(* Logix 5000 project; controller RG_Chopper vendor 1 type 14 code 235 rev 32.12; software revision 32.04; part 4 of 6 *)
(* tags used below, declared in another part *)
   L2_FAIL_TMR : TIMER;   // LSSL2 Fail Always Open Detect
   LSSL2_FAIL : BOOL;   // Lower Safety Limit Switch LSS-L2 Fail
   LSSL2_FAIL2 : BOOL;   // Lower Safety Limit Switch LSS-L2 Mode 2
   LSSU2_FAIL : BOOL;   // Upper Safety Limit Switch LSS-U2 Fail
   LSSU2_FAIL2 : BOOL;   // Upper Safety Limit Switch USS-L2 Mode 2
   U2_FAIL_TMR : TIMER;   // LSSU2 Fail Always Open Detect
   _DBL101_TANK_LEVEL : BOOL;   // Conentrate Chopper Level Switch Local:1:I.Data.9
   ALARM_FATAL : BOOL;   // Fatal Alarm Stops All Operation
   ALARM_GATE_OPEN : BOOL;   // Gate Open
   AUTO_ALL : BOOL;   // All Devices to AUTO
   CB104_DUMPER_AUX : BOOL;   // CB104 Dumper Aux From Dumper Control
   CIP_CMPLT : BOOL;   // CIP Complete Indicator
   CYC_CIP : BOOL;   // CIP Cycle Running
   CYC_RUN : BOOL;   // Production Cycle Running
   DBT101 : TD_TA_TP_8PORT_IOL;   // DTT101 Hot Water Temperature IO-Link RAW
   DBT102 : TD_TA_TP_8PORT_IOL;   // DBT102 Product Temperature IO-Link RAW
   DBX101_AM : PUSH_PUSH_PB;   // DBX-101 Push-Push Button Control
   DBX101_AUX : BOOL;   // DBX-101 Agitator Motor Aux
   DBX101_CTL : HOA_CTRL_v2;   // DBX-101 Agitator Motor Control Block
   DBX101_FAULT : BOOL;
   DBX101_MAN : PUSH_PUSH_PB;   // DBX-101 Manual Run Push-Push
   DBX101_OL : BOOL;   // DBX-101 Motor OverLoad Status
   DBX101_START : BOOL;   // DBX-101 Agitator Start Safety Mapped DBX101_S_START
   DBX102_AM : PUSH_PUSH_PB;   // DBX-102 Push-Push Button Control
   DBX102_AUX : ALIAS FOR SIGNAL_IN_RG_CHOPPER.0;   // DBX-102 VFD Active AUX
   DBX102_CTL : HOA_CTRL_v2;   // DBX102 Product Discharge Pump Control Block
   DBX102_FAULT : BOOL;   // DBX-102 Discharge Pump Drive Fault
   DBX102_M_FAULT : BOOL;   // DBX-102 Discharge Pump Drive or Motor Fault
   DBX102_MAN : PUSH_PUSH_PB;   // DBX-102 Manual Control Push-Push
   DBX102_START : BOOL;   // DBX-102 Product Pump VFD START
   DBX103_AM : PUSH_PUSH_PB;   // DBX-103 Push-Push Button Control
   DBX103_AUX : BOOL;   // DBX-103 Water Pump Aux
   DBX103_CTL : HOA_CTRL_v2;   // DBX-103 Hot Water Pump Control Block
   DBX103_FAULT : BOOL;   // DBX-103 Hot Water Pump Fault
   DBX103_MAN : PUSH_PUSH_PB;   // DBX-103 Manual Run Push-Push
   DBX103_OL : BOOL;   // DBX-103 Motor OverLoad Status
   DBX103_START : BOOL;   // DBX-103 Water Pump Start Safety Mapped DBX103_S_START
   DBX104_AM : PUSH_PUSH_PB;   // DBX-104 Push-Push Button Control
   DBX104_AUX : BOOL;   // DBX-104 VFD Active AUX
   DBX104_CTL : HOA_CTRL_v2;   // DBX-104 Reversing Motor Starter Control
   DBX104_DD : PUSH_PUSH_PB;   // DBX104 VFD Direction DOWN Control
   DBX104_DU : PUSH_PUSH_PB;   // DBX104 VFD Direction UP Control
   DBX104_DWN : BOOL;   // DBX-104 Drum Dumper VFD Direction DOWN
   DBX104_FAULT : BOOL;   // DBX-104 Dumper Elevator Drive Fault
   DBX104_M_FAULT : BOOL;   // DBX-104 Dumper Elevator Drive or Motor Fault
   DBX104_MAN : PUSH_PUSH_PB;   // DBX-104 Manual Control Push-Push
   DBX104_START : BOOL;   // DBX-104 Drum Dumper VFD START
   DBX104_UP : BOOL;   // DBX-104 Drum Dumper VFD Direction UP
   DLT101 : PN_PI_PP_8PORT_IOL;   // DLT101 Tank Level IO-Link RAW
   DLT101_LVL_SCL : REAL;   // Tank Level Scaled (0.0 - 100.0%)
   DLT101_SCL : ANLG_SCALE;   // Tank Level Scaling Block
   DLT101_Tk : TK_CTRL;   // Tank Level Control
   DTT101 : REAL;   // DTT-101 Hot Water Temperature Analong In
   DTT102 : REAL;   // Discharge Product Temperature
   DWN_MKBK : BOOL;   // Elevator Down Make / Break LS_L1 Detection
   DWN_MKBK1 : BOOL;   // Elevator Down Make / Break Memory 1
   DWN_STP : BOOL;   // Elevator Down STOP
   Fault_ACK : BOOL;   // Fault Acknowledge
   FAULT_ACK_PB : BOOL;   // Fault ACK Push Button
   Gate_SW1 : DCI_MONITOR;   // Safety Switch Gate_SW1 SW105 A/B
   Gate_SW2 : DCI_MONITOR;   // Safety Switch Gate_SW2 SW108 A/B
   LEVEL_TIMER : TIMER;   // Juice Tank At High Level
   LOT1_TMR : TIMER;   // Lower Over Travel Switch Disable Timer
   LS_L1 : BOOL;   // New Dumper LOWER Limit Switch #1
   LS_LID_OPN : BOOL;   // Lid Open Switch IO-Link Master Mapped X04
   LS_M1 : BOOL;   // New Dumper MIDDLE Limit Switch #1
   LS_U1 : BOOL;   // New Dumper UPPER Limit Switch #1
   LSS_L2 : BOOL;   // New Dumper LOWER Safety Limit Switch #2
   LSS_LOT1 : BOOL;   // New Dumper LOWER OVER TRAVEL Limit Switch
   LSS_U2 : BOOL;   // New Dumper UPPER Safety Limit Switch #2
   ONESHOT : DINT;   // One-shot Word
   PB101 : BOOL;   // Drum Dumper Elevator UP Push Button
   PB102 : BOOL;   // Drum Dumper Elevator DOWN Push Button
   PB103 : BOOL;   // Drum Dumper Elevator STOP Push Button
   PROC_TMR : TIMER[16];   // Process Timers
   S_ESTOP : BOOL;   // Safety ESTOP
   S_Fault_Res : BOOL;   // Safety Circuit Fault Reset
   S_SW_IN : DINT;   // Safety Switch Input Array
   SCR1291 : BOOL;   // Dumper Estop Permissive Lost SCR-1291
   SHTDWN_ACTV : BOOL;   // System Shutdown is In Progress
   SHTDWN_CMPLT : BOOL;   // System Shutdown Complete
   SHUTDOWN : DINT;   // System Shutdown Control Bits
   SIGNAL_OUT_RG_CHOPPER : DINT;
   SPARE_IN : DINT;   // Spare Input
   STARTUP : DINT;   // System Startup Control Bits
   STOP_ALL : BOOL;   // Stop All
   SW101_START_PB : BOOL;   // Start PB HMI
   SW102_STOP_PB : BOOL;   // Stop PB HMI
   SW103_CIP_PB : BOOL;   // CIP PB HMI
   SW104_ESTOP : BOOL;   // Safety E-Stop SW-104
   SW105_DEBOUNCE : TIMER;   // SW-105 Gate Switch Debounce Timer
   SW105_GATE_SWITCH : BOOL;   // Safety Switch Gate SW #1 SW105 A/B
   SW106_LC : LIGHT_CURTAIN;   // Safety SW106 Light Curain
   SW106_LIGHT_CUR : BOOL;   // Safety Light Curtain SW-106
   SW107_TANK_LID : BOOL;   // Tank Lid Safety Switch Active
   SW108_DEBOUNCE : TIMER;   // SW-108 Gate Switch Debounce Timer
   SW108_GATE_SWITCH : BOOL;   // Safety Switch Gate SW #2 SW108 A/B
   SW109 : BOOL;   // Drum Dumper Upper Limit Switch
   SW110 : BOOL;   // Drum Dumper Lower Limit Switch
   Tank_Lid1 : EMERGENCY_STOP;   // Safety Switch Tank Lid Status SW105 A/B
   TP3232_TMP_1_Scaled : REAL;   // Hot Water Temperature Scaled
   TP3232_TMP_2_Scaled : REAL;   // Product Temperature Scaled
   UP_MKBK : BOOL;   // Elevator Down Make / Break LS_U1 Detection
   UP_MKBK1 : BOOL;   // Elevator Up Make / Break Memory 1
   UP_STP : BOOL;   // Elevator Up STOP
(* MainProgram, continued *)

ROUTINE InLink   (* ladder *)
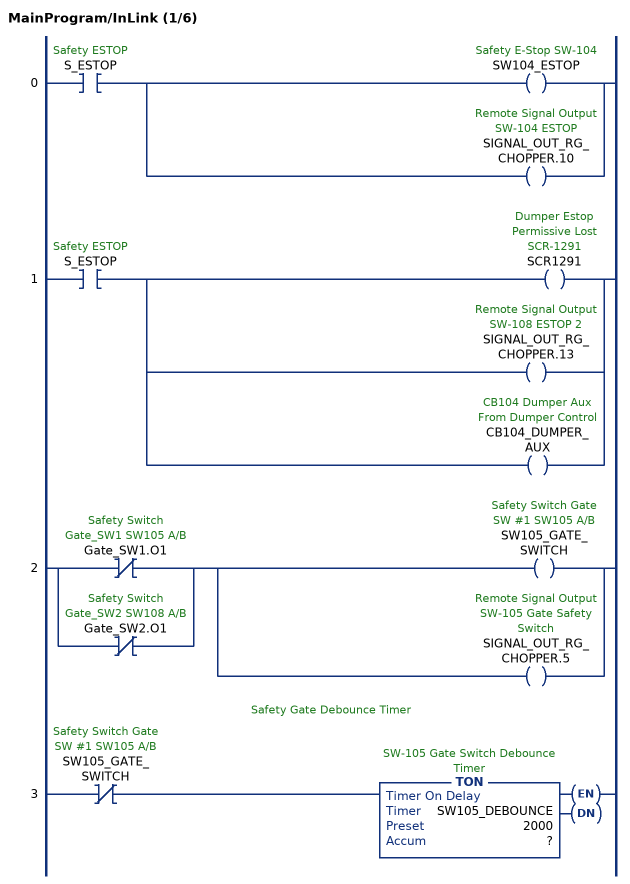
   0: XIC(S_ESTOP)[OTE(SW104_ESTOP) ,OTE(SIGNAL_OUT_RG_CHOPPER.10) ];
   1: XIC(S_ESTOP)[OTE(SCR1291) ,OTE(SIGNAL_OUT_RG_CHOPPER.13) ,OTE(CB104_DUMPER_AUX) ];
   2: [XIO(Gate_SW1.O1) ,XIO(Gate_SW2.O1) ][OTE(SW105_GATE_SWITCH) ,OTE(SIGNAL_OUT_RG_CHOPPER.5) ];
   // Safety Gate Debounce Timer
   3: XIO(SW105_GATE_SWITCH)TON(SW105_DEBOUNCE,?,?);
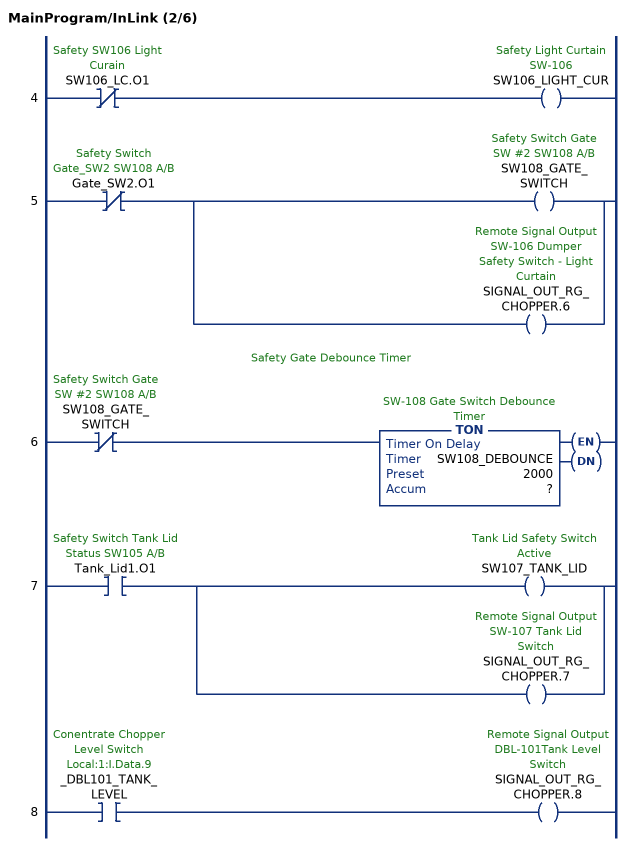
   4: XIO(SW106_LC.O1)OTE(SW106_LIGHT_CUR);
   5: XIO(Gate_SW2.O1)[OTE(SW108_GATE_SWITCH) ,OTE(SIGNAL_OUT_RG_CHOPPER.6) ];
   // Safety Gate Debounce Timer
   6: XIO(SW108_GATE_SWITCH)TON(SW108_DEBOUNCE,?,?);
   7: XIC(Tank_Lid1.O1)[OTE(SW107_TANK_LID) ,OTE(SIGNAL_OUT_RG_CHOPPER.7) ];
   8: XIC(_DBL101_TANK_LEVEL)OTE(SIGNAL_OUT_RG_CHOPPER.8);
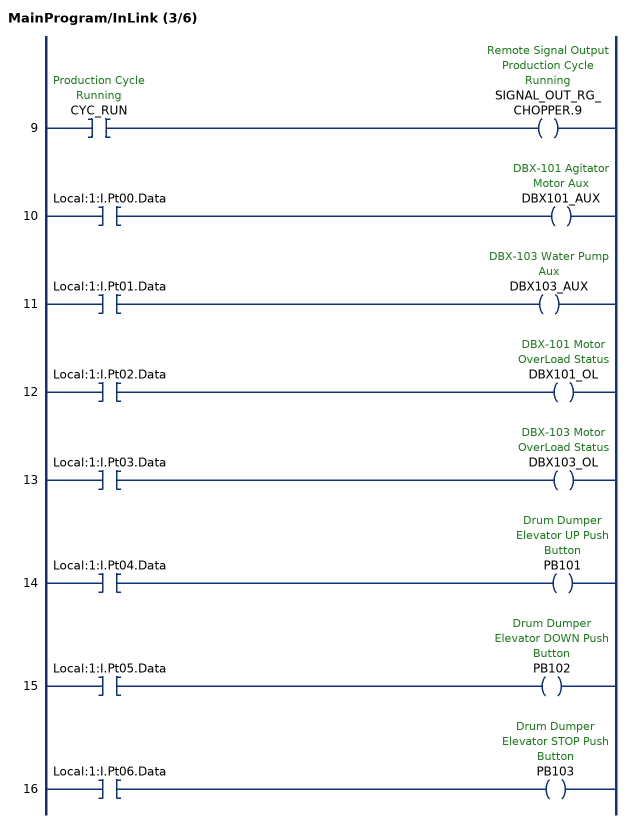
   9: XIC(CYC_RUN)OTE(SIGNAL_OUT_RG_CHOPPER.9);
   10: XIC(Local:1:I.Pt00.Data)OTE(DBX101_AUX);
   11: XIC(Local:1:I.Pt01.Data)OTE(DBX103_AUX);
   12: XIC(Local:1:I.Pt02.Data)OTE(DBX101_OL);
   13: XIC(Local:1:I.Pt03.Data)OTE(DBX103_OL);
   14: XIC(Local:1:I.Pt04.Data)OTE(PB101);
   15: XIC(Local:1:I.Pt05.Data)OTE(PB102);
   16: XIC(Local:1:I.Pt06.Data)OTE(PB103);
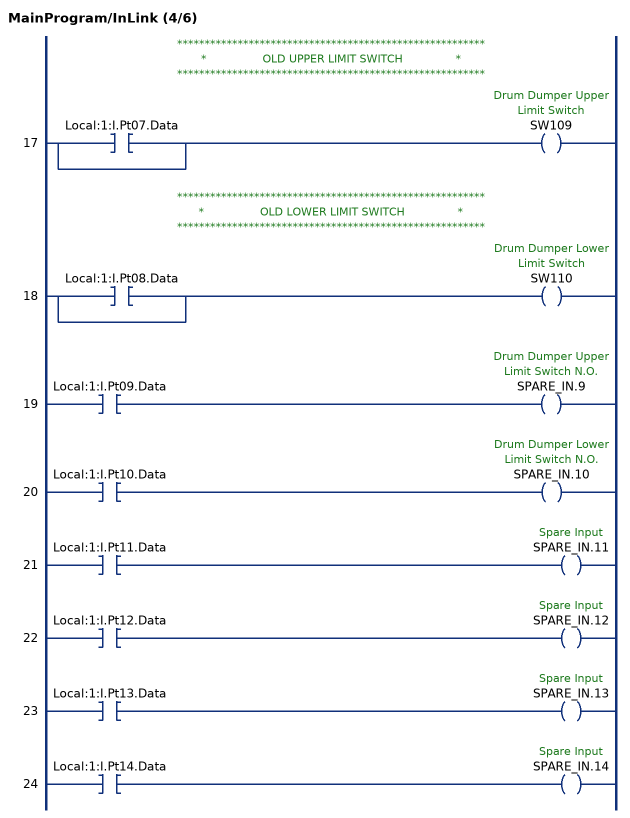
   // ********************************************************
   // *                OLD UPPER LIMIT SWITCH               *
   // ********************************************************
   17: [XIC(Local:1:I.Pt07.Data) ,]OTE(SW109);
   // ********************************************************
   // *                OLD LOWER LIMIT SWITCH               *
   // ********************************************************
   18: [XIC(Local:1:I.Pt08.Data) ,]OTE(SW110);
   19: XIC(Local:1:I.Pt09.Data)OTE(SPARE_IN.9);
   20: XIC(Local:1:I.Pt10.Data)OTE(SPARE_IN.10);
   21: XIC(Local:1:I.Pt11.Data)OTE(SPARE_IN.11);
   22: XIC(Local:1:I.Pt12.Data)OTE(SPARE_IN.12);
   23: XIC(Local:1:I.Pt13.Data)OTE(SPARE_IN.13);
   24: XIC(Local:1:I.Pt14.Data)OTE(SPARE_IN.14);
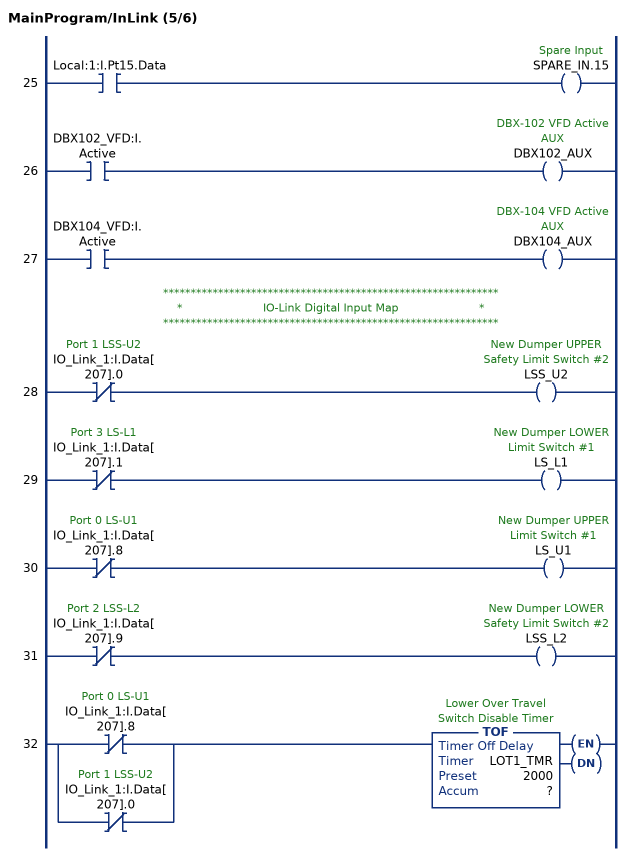
   25: XIC(Local:1:I.Pt15.Data)OTE(SPARE_IN.15);
   26: XIC(DBX102_VFD:I.Active)OTE(DBX102_AUX);
   27: XIC(DBX104_VFD:I.Active)OTE(DBX104_AUX);
   // *************************************************************
   // *                       IO-Link Digital Input Map                       *
   // *************************************************************
   28: XIO(IO_Link_1:I.Data[207].0)OTE(LSS_U2);
   29: XIO(IO_Link_1:I.Data[207].1)OTE(LS_L1);
   30: XIO(IO_Link_1:I.Data[207].8)OTE(LS_U1);
   31: XIO(IO_Link_1:I.Data[207].9)OTE(LSS_L2);
   32: [XIO(IO_Link_1:I.Data[207].8) ,XIO(IO_Link_1:I.Data[207].0) ]TOF(LOT1_TMR,?,?);
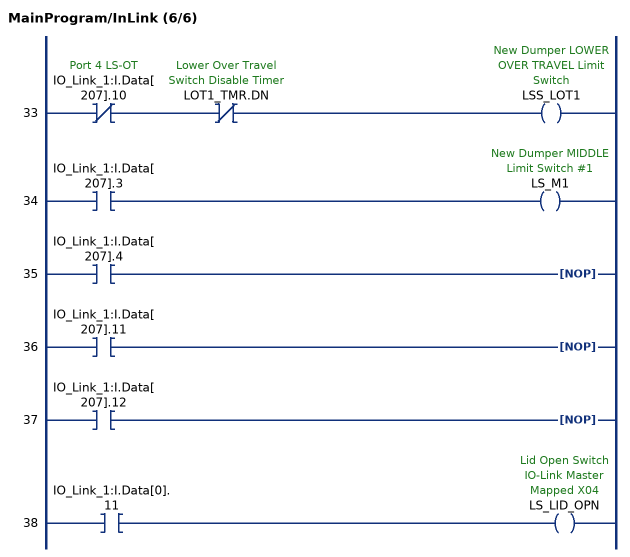
   33: XIO(IO_Link_1:I.Data[207].10)XIO(LOT1_TMR.DN)OTE(LSS_LOT1);
   34: XIC(IO_Link_1:I.Data[207].3)OTE(LS_M1);
   35: XIC(IO_Link_1:I.Data[207].4)NOP();
   36: XIC(IO_Link_1:I.Data[207].11)NOP();
   37: XIC(IO_Link_1:I.Data[207].12)NOP();
   38: XIC(IO_Link_1:I.Data[0].11)OTE(LS_LID_OPN);
END_ROUTINE

ROUTINE IO_Link   (* ladder *)
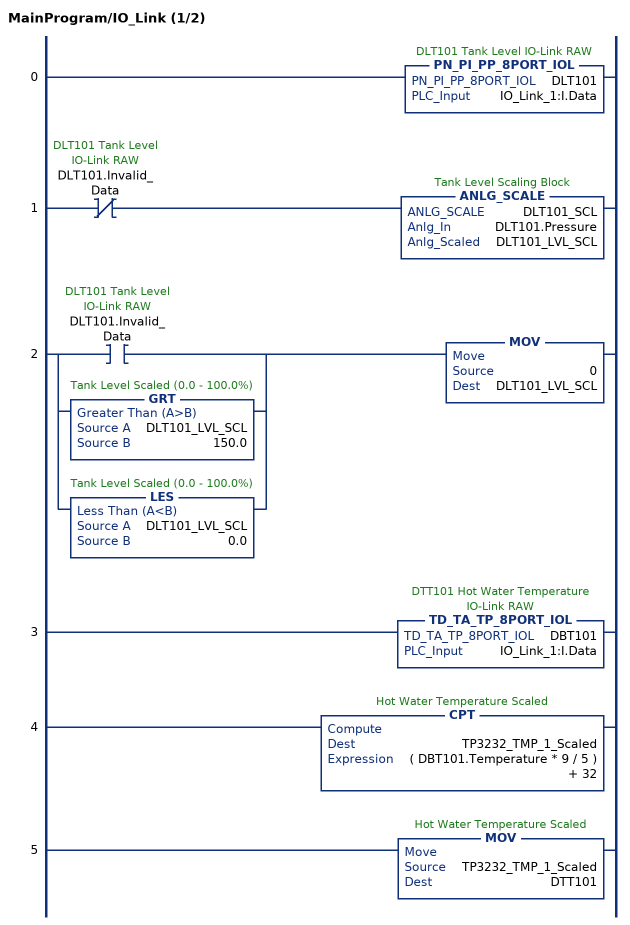
   0: PN_PI_PP_8PORT_IOL(DLT101,IO_Link_1:I.Data);
   1: XIO(DLT101.Invalid_Data)ANLG_SCALE(DLT101_SCL,DLT101.Pressure,DLT101_LVL_SCL);
   2: [XIC(DLT101.Invalid_Data) ,GRT(DLT101_LVL_SCL,150.0) ,LES(DLT101_LVL_SCL,0.0) ]MOV(0,DLT101_LVL_SCL);
   3: TD_TA_TP_8PORT_IOL(DBT101,IO_Link_1:I.Data);
   4: CPT(TP3232_TMP_1_Scaled,( DBT101.Temperature * 9 / 5 ) + 32);
   5: MOV(TP3232_TMP_1_Scaled,DTT101);
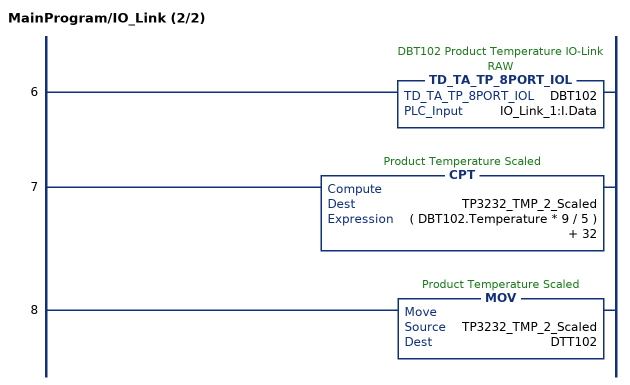
   6: TD_TA_TP_8PORT_IOL(DBT102,IO_Link_1:I.Data);
   7: CPT(TP3232_TMP_2_Scaled,( DBT102.Temperature * 9 / 5 ) + 32);
   8: MOV(TP3232_TMP_2_Scaled,DTT102);
END_ROUTINE

ROUTINE LOGIC   (* ladder *)
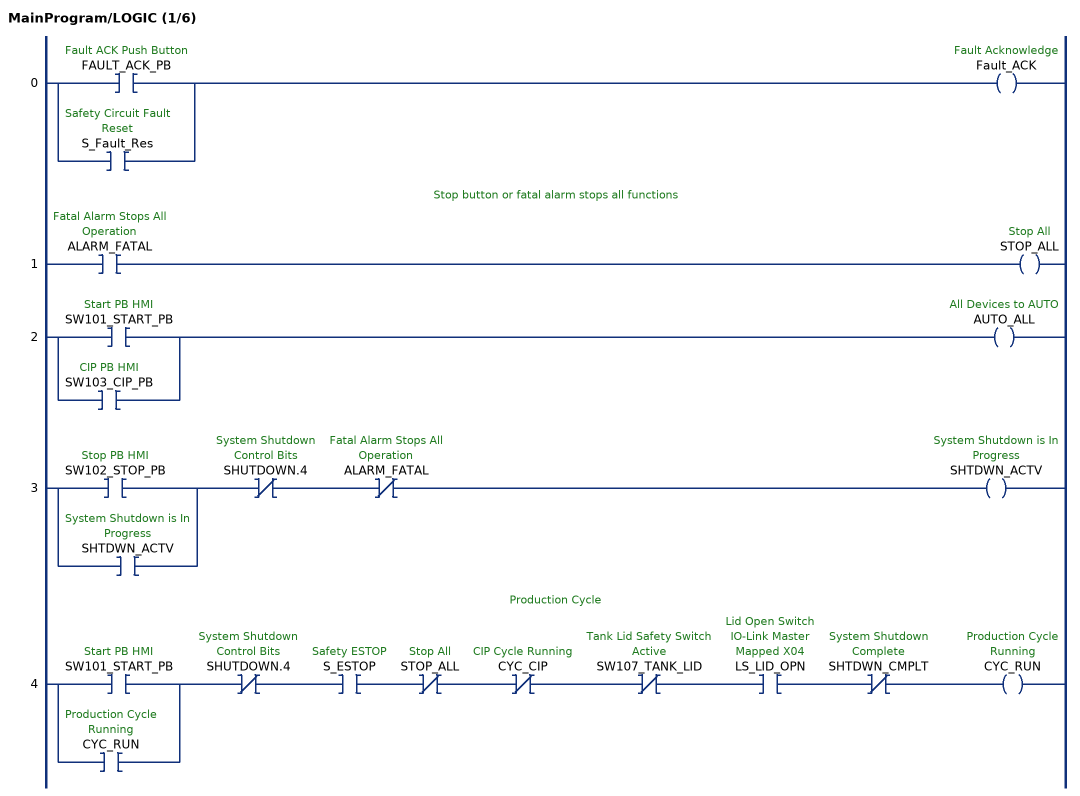
   0: [XIC(FAULT_ACK_PB) ,XIC(S_Fault_Res) ]OTE(Fault_ACK);
   // Stop button or fatal alarm stops all functions
   1: XIC(ALARM_FATAL)OTE(STOP_ALL);
   2: [XIC(SW101_START_PB) ,XIC(SW103_CIP_PB) ]OTE(AUTO_ALL);
   3: [XIC(SW102_STOP_PB) ,XIC(SHTDWN_ACTV) ]XIO(SHUTDOWN.4)XIO(ALARM_FATAL)OTE(SHTDWN_ACTV);
   // Production Cycle
   4: [XIC(SW101_START_PB) ,XIC(CYC_RUN) ]XIO(SHUTDOWN.4)XIC(S_ESTOP)XIO(STOP_ALL)XIO(CYC_CIP)XIO(SW107_TANK_LID)XIC(LS_LID_OPN)XIO(SHTDWN_CMPLT)OTE(CYC_RUN);
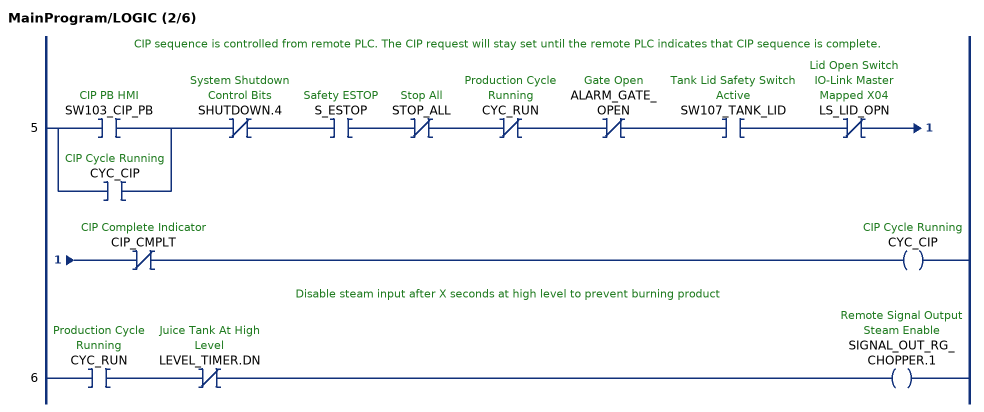
   // CIP sequence is controlled from remote PLC. The CIP request will stay set until the remote PLC indicates that CIP sequence is complete.
   5: [XIC(SW103_CIP_PB) ,XIC(CYC_CIP) ]XIO(SHUTDOWN.4)XIC(S_ESTOP)XIO(STOP_ALL)XIO(CYC_RUN)XIO(ALARM_GATE_OPEN)XIC(SW107_TANK_LID)XIO(LS_LID_OPN)XIO(CIP_CMPLT)OTE(CYC_CIP);
   // Disable steam input after X seconds at high level to prevent burning product
   6: XIC(CYC_RUN)XIO(LEVEL_TIMER.DN)OTE(SIGNAL_OUT_RG_CHOPPER.1);
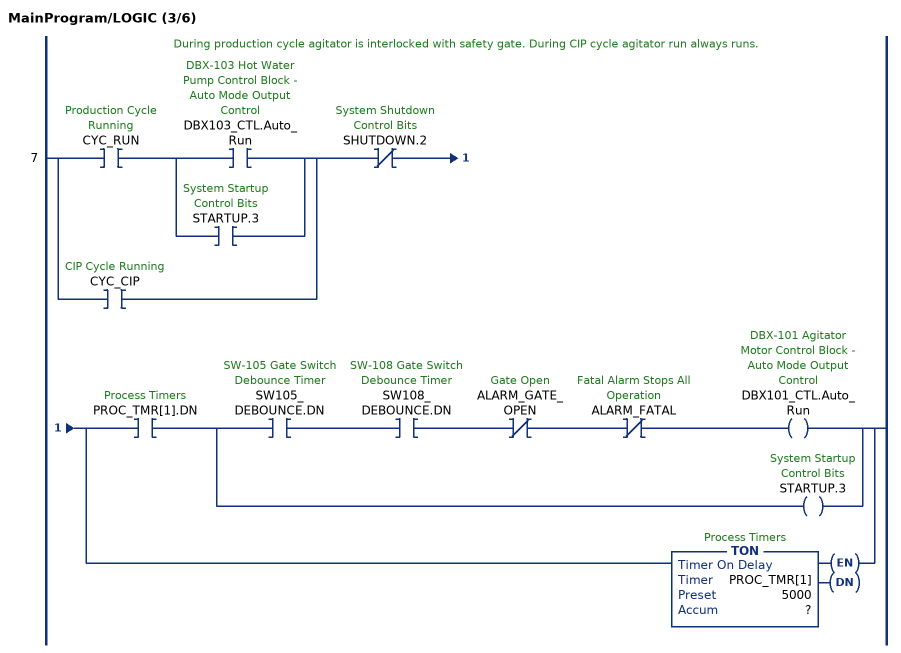
   // During production cycle agitator is interlocked with safety gate. During CIP cycle agitator run always runs.
   7: [XIC(CYC_RUN) [XIC(DBX103_CTL.Auto_Run) ,XIC(STARTUP.3) ] ,XIC(CYC_CIP) ]XIO(SHUTDOWN.2)[XIC(PROC_TMR[1].DN) [XIC(SW105_DEBOUNCE.DN) XIC(SW108_DEBOUNCE.DN) XIO(ALARM_GATE_OPEN) XIO(ALARM_FATAL) OTE(DBX101_CTL.Auto_Run) ,OTE(STARTUP.3) ] ,TON(PROC_TMR[1],?,?) ];
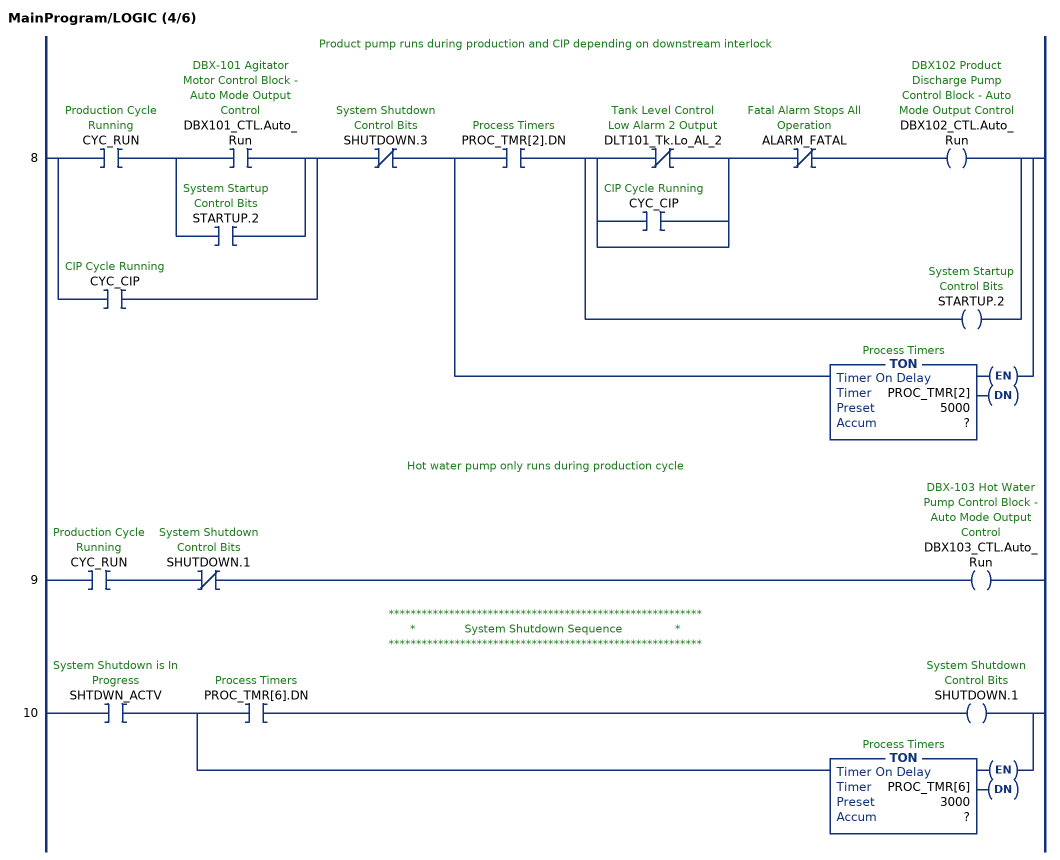
   // Product pump runs during production and CIP depending on downstream interlock
   8: [XIC(CYC_RUN) [XIC(DBX101_CTL.Auto_Run) ,XIC(STARTUP.2) ] ,XIC(CYC_CIP) ]XIO(SHUTDOWN.3)[XIC(PROC_TMR[2].DN) [[XIO(DLT101_Tk.Lo_AL_2) ,XIC(CYC_CIP) ,] XIO(ALARM_FATAL) OTE(DBX102_CTL.Auto_Run) ,OTE(STARTUP.2) ] ,TON(PROC_TMR[2],?,?) ];
   // Hot water pump only runs during production cycle
   9: XIC(CYC_RUN)XIO(SHUTDOWN.1)OTE(DBX103_CTL.Auto_Run);
   // *********************************************************
   // *              System Shutdown Sequence               *
   // *********************************************************
   10: XIC(SHTDWN_ACTV)[XIC(PROC_TMR[6].DN) OTE(SHUTDOWN.1) ,TON(PROC_TMR[6],?,?) ];
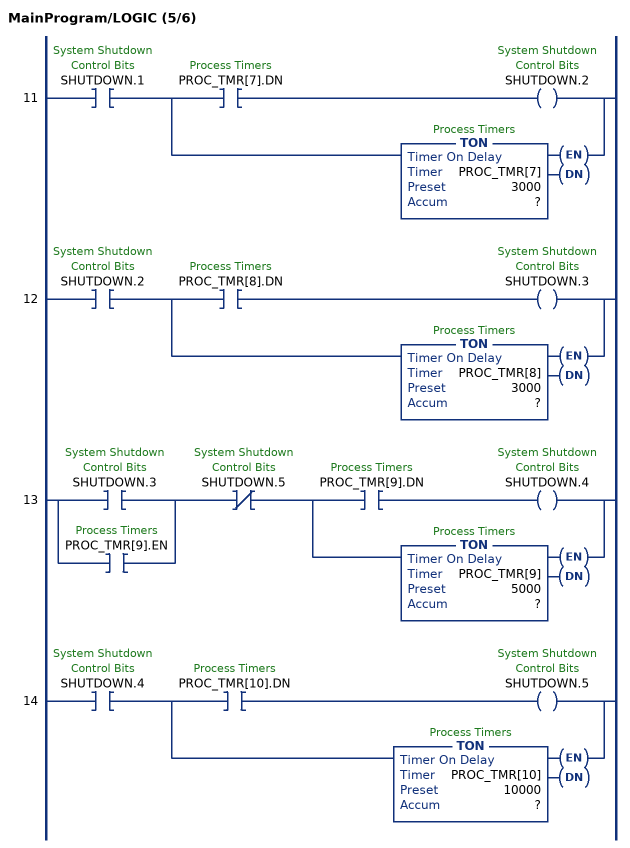
   11: XIC(SHUTDOWN.1)[XIC(PROC_TMR[7].DN) OTE(SHUTDOWN.2) ,TON(PROC_TMR[7],?,?) ];
   12: XIC(SHUTDOWN.2)[XIC(PROC_TMR[8].DN) OTE(SHUTDOWN.3) ,TON(PROC_TMR[8],?,?) ];
   13: [XIC(SHUTDOWN.3) ,XIC(PROC_TMR[9].EN) ]XIO(SHUTDOWN.5)[XIC(PROC_TMR[9].DN) OTE(SHUTDOWN.4) ,TON(PROC_TMR[9],?,?) ];
   14: XIC(SHUTDOWN.4)[XIC(PROC_TMR[10].DN) OTE(SHUTDOWN.5) ,TON(PROC_TMR[10],?,?) ];
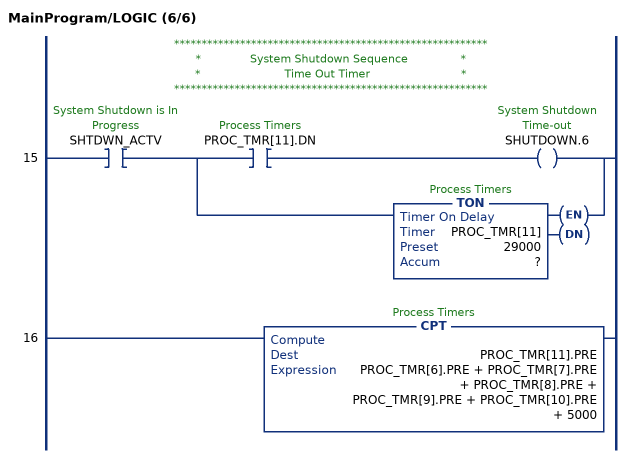
   // *********************************************************
   // *              System Shutdown Sequence               *
   // *                        Time Out Timer                          *
   // *********************************************************
   15: XIC(SHTDWN_ACTV)[XIC(PROC_TMR[11].DN) OTE(SHUTDOWN.6) ,TON(PROC_TMR[11],?,?) ];
   16: CPT(PROC_TMR[11].PRE,PROC_TMR[6].PRE + PROC_TMR[7].PRE + PROC_TMR[8].PRE + PROC_TMR[9].PRE + PROC_TMR[10].PRE + 5000);
END_ROUTINE

ROUTINE MainRoutine   (* ladder *)
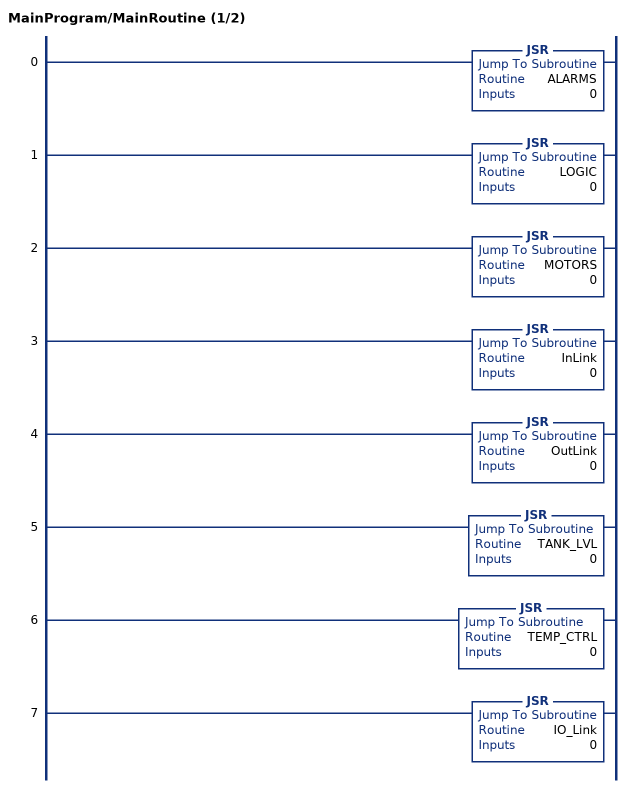
   0: JSR(ALARMS,0);
   1: JSR(LOGIC,0);
   2: JSR(MOTORS,0);
   3: JSR(InLink,0);
   4: JSR(OutLink,0);
   5: JSR(TANK_LVL,0);
   6: JSR(TEMP_CTRL,0);
   7: JSR(IO_Link,0);
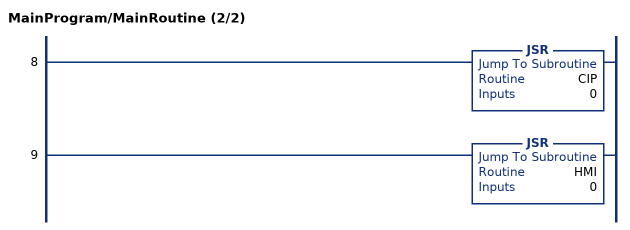
   8: JSR(CIP,0);
   9: JSR(HMI,0);
END_ROUTINE

ROUTINE MOTORS   (* ladder *)
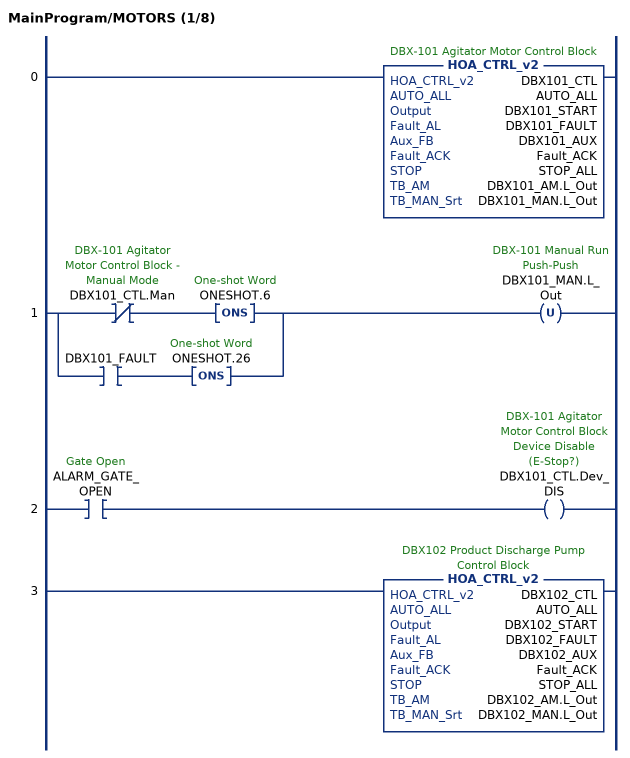
   0: HOA_CTRL_v2(DBX101_CTL,AUTO_ALL,DBX101_START,DBX101_FAULT,DBX101_AUX,Fault_ACK,STOP_ALL,DBX101_AM.L_Out,DBX101_MAN.L_Out);
   1: [XIO(DBX101_CTL.Man) ONS(ONESHOT.6) ,XIC(DBX101_FAULT) ONS(ONESHOT.26) ]OTU(DBX101_MAN.L_Out);
   2: XIC(ALARM_GATE_OPEN)OTE(DBX101_CTL.Dev_DIS);
   3: HOA_CTRL_v2(DBX102_CTL,AUTO_ALL,DBX102_START,DBX102_FAULT,DBX102_AUX,Fault_ACK,STOP_ALL,DBX102_AM.L_Out,DBX102_MAN.L_Out);
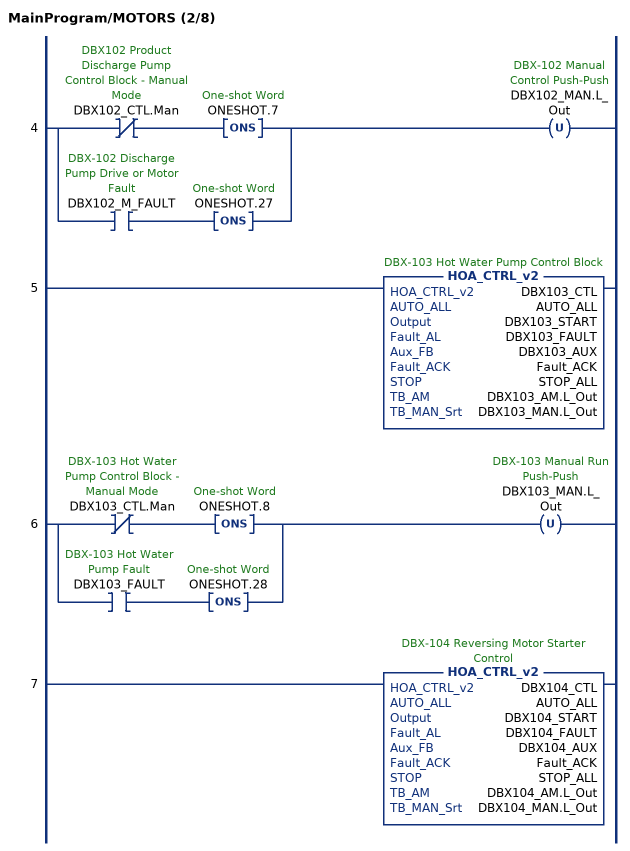
   4: [XIO(DBX102_CTL.Man) ONS(ONESHOT.7) ,XIC(DBX102_M_FAULT) ONS(ONESHOT.27) ]OTU(DBX102_MAN.L_Out);
   5: HOA_CTRL_v2(DBX103_CTL,AUTO_ALL,DBX103_START,DBX103_FAULT,DBX103_AUX,Fault_ACK,STOP_ALL,DBX103_AM.L_Out,DBX103_MAN.L_Out);
   6: [XIO(DBX103_CTL.Man) ONS(ONESHOT.8) ,XIC(DBX103_FAULT) ONS(ONESHOT.28) ]OTU(DBX103_MAN.L_Out);
   7: HOA_CTRL_v2(DBX104_CTL,AUTO_ALL,DBX104_START,DBX104_FAULT,DBX104_AUX,Fault_ACK,STOP_ALL,DBX104_AM.L_Out,DBX104_MAN.L_Out);
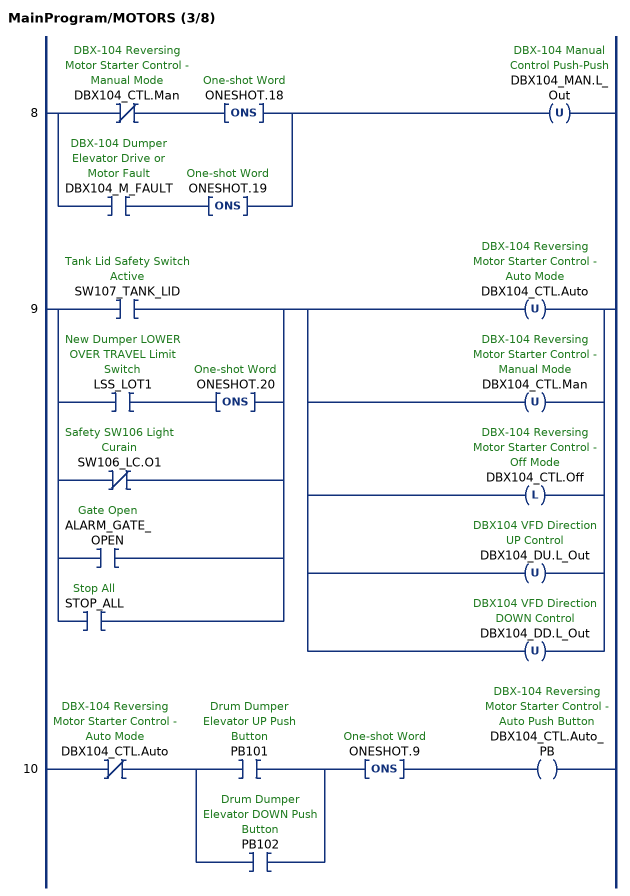
   8: [XIO(DBX104_CTL.Man) ONS(ONESHOT.18) ,XIC(DBX104_M_FAULT) ONS(ONESHOT.19) ]OTU(DBX104_MAN.L_Out);
   9: [XIC(SW107_TANK_LID) ,XIC(LSS_LOT1) ONS(ONESHOT.20) ,XIO(SW106_LC.O1) ,XIC(ALARM_GATE_OPEN) ,XIC(STOP_ALL) ][OTU(DBX104_CTL.Auto) ,OTU(DBX104_CTL.Man) ,OTL(DBX104_CTL.Off) ,OTU(DBX104_DU.L_Out) ,OTU(DBX104_DD.L_Out) ];
   10: XIO(DBX104_CTL.Auto)[XIC(PB101) ,XIC(PB102) ]ONS(ONESHOT.9)OTE(DBX104_CTL.Auto_PB);
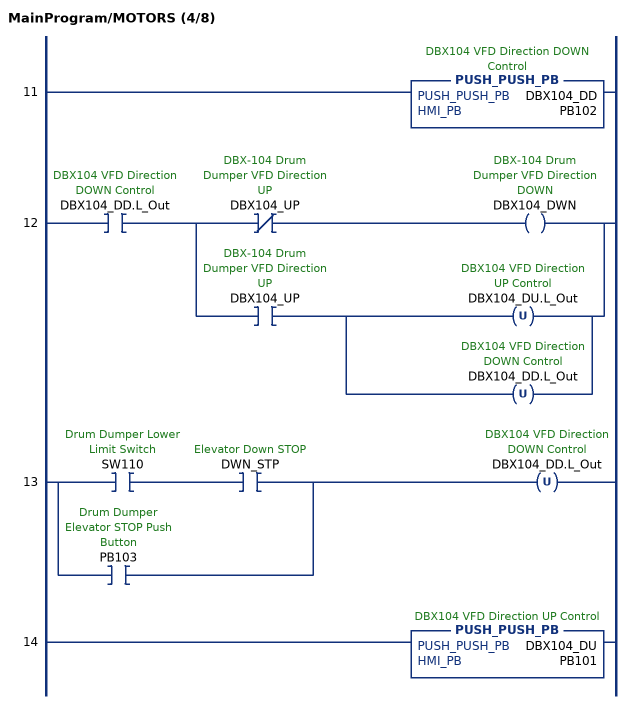
   11: PUSH_PUSH_PB(DBX104_DD,PB102);
   12: XIC(DBX104_DD.L_Out)[XIO(DBX104_UP) OTE(DBX104_DWN) ,XIC(DBX104_UP) [OTU(DBX104_DU.L_Out) ,OTU(DBX104_DD.L_Out) ] ];
   13: [XIC(SW110) XIC(DWN_STP) ,XIC(PB103) ]OTU(DBX104_DD.L_Out);
   14: PUSH_PUSH_PB(DBX104_DU,PB101);
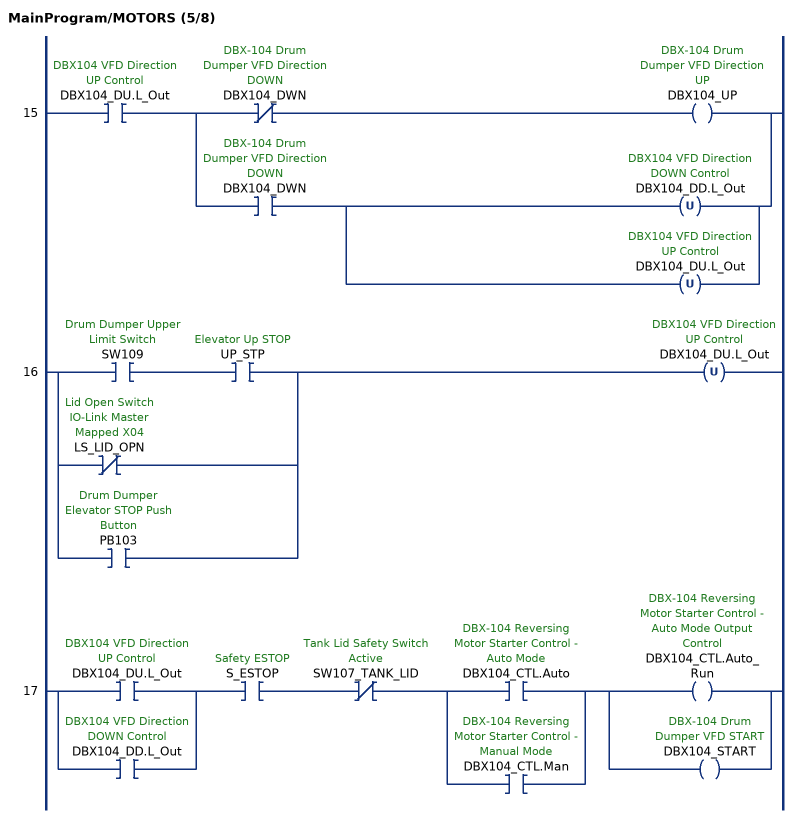
   15: XIC(DBX104_DU.L_Out)[XIO(DBX104_DWN) OTE(DBX104_UP) ,XIC(DBX104_DWN) [OTU(DBX104_DD.L_Out) ,OTU(DBX104_DU.L_Out) ] ];
   16: [XIC(SW109) XIC(UP_STP) ,XIO(LS_LID_OPN) ,XIC(PB103) ]OTU(DBX104_DU.L_Out);
   17: [XIC(DBX104_DU.L_Out) ,XIC(DBX104_DD.L_Out) ]XIC(S_ESTOP)XIO(SW107_TANK_LID)[XIC(DBX104_CTL.Auto) ,XIC(DBX104_CTL.Man) ][OTE(DBX104_CTL.Auto_Run) ,OTE(DBX104_START) ];
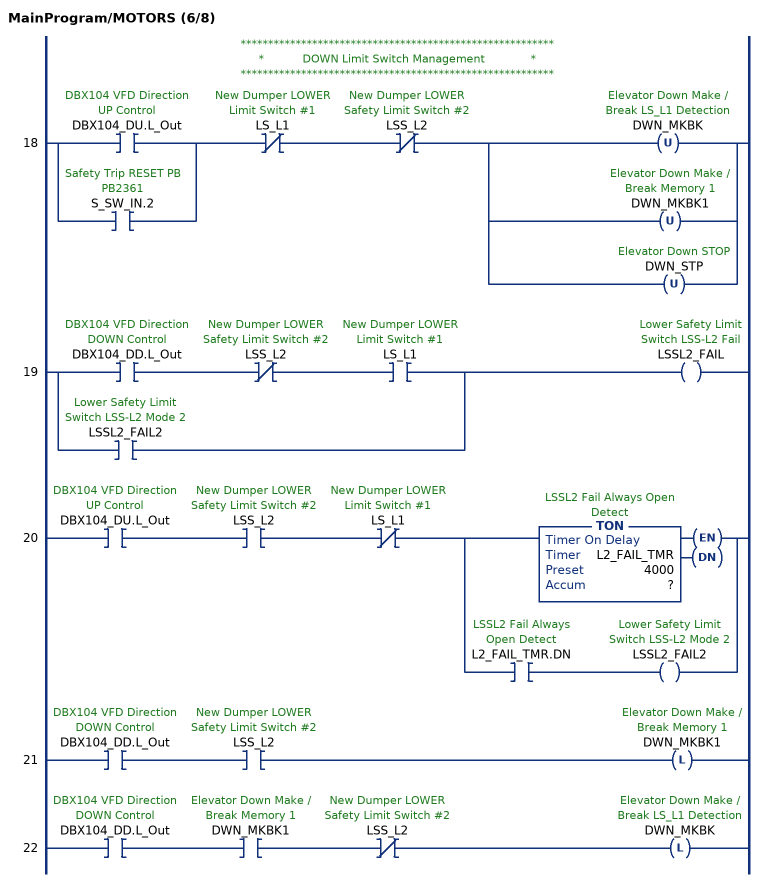
   // *********************************************************
   // *           DOWN Limit Switch Management             *
   // *********************************************************
   18: [XIC(DBX104_DU.L_Out) ,XIC(S_SW_IN.2) ]XIO(LS_L1)XIO(LSS_L2)[OTU(DWN_MKBK) ,OTU(DWN_MKBK1) ,OTU(DWN_STP) ];
   19: [XIC(DBX104_DD.L_Out) XIO(LSS_L2) XIC(LS_L1) ,XIC(LSSL2_FAIL2) ]OTE(LSSL2_FAIL);
   20: XIC(DBX104_DU.L_Out)XIC(LSS_L2)XIO(LS_L1)[TON(L2_FAIL_TMR,?,?) ,XIC(L2_FAIL_TMR.DN) OTE(LSSL2_FAIL2) ];
   21: XIC(DBX104_DD.L_Out)XIC(LSS_L2)OTL(DWN_MKBK1);
   22: XIC(DBX104_DD.L_Out)XIC(DWN_MKBK1)XIO(LSS_L2)OTL(DWN_MKBK);
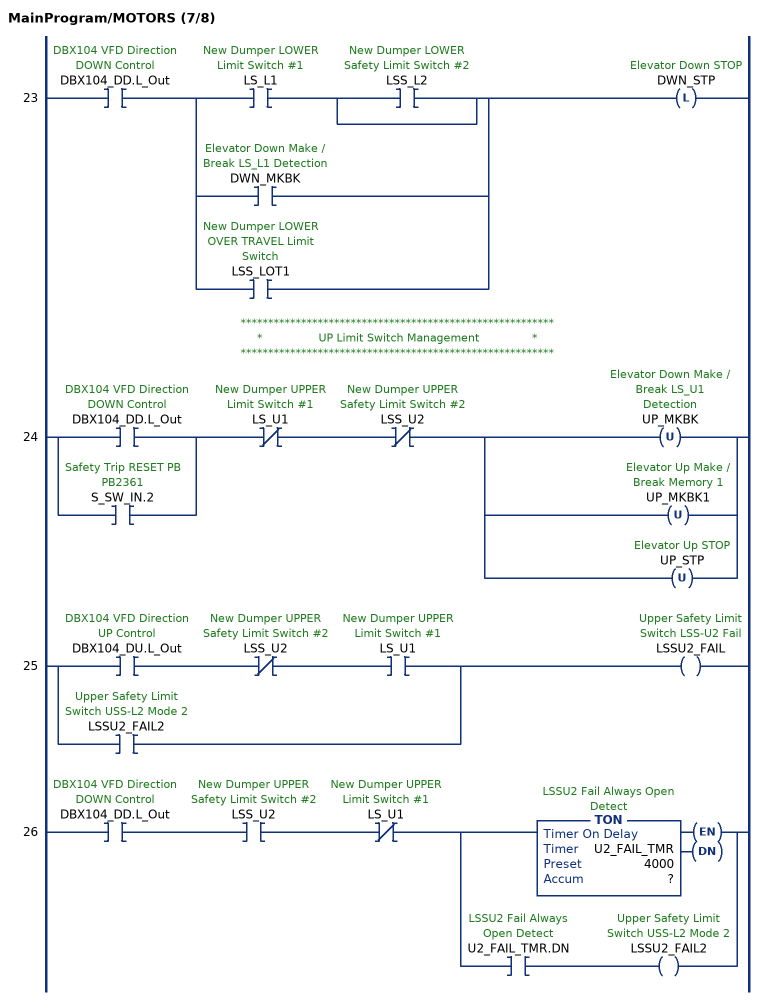
   23: XIC(DBX104_DD.L_Out)[XIC(LS_L1) [XIC(LSS_L2) ,] ,XIC(DWN_MKBK) ,XIC(LSS_LOT1) ]OTL(DWN_STP);
   // *********************************************************
   // *                UP Limit Switch Management               *
   // *********************************************************
   24: [XIC(DBX104_DD.L_Out) ,XIC(S_SW_IN.2) ]XIO(LS_U1)XIO(LSS_U2)[OTU(UP_MKBK) ,OTU(UP_MKBK1) ,OTU(UP_STP) ];
   25: [XIC(DBX104_DU.L_Out) XIO(LSS_U2) XIC(LS_U1) ,XIC(LSSU2_FAIL2) ]OTE(LSSU2_FAIL);
   26: XIC(DBX104_DD.L_Out)XIC(LSS_U2)XIO(LS_U1)[TON(U2_FAIL_TMR,?,?) ,XIC(U2_FAIL_TMR.DN) OTE(LSSU2_FAIL2) ];
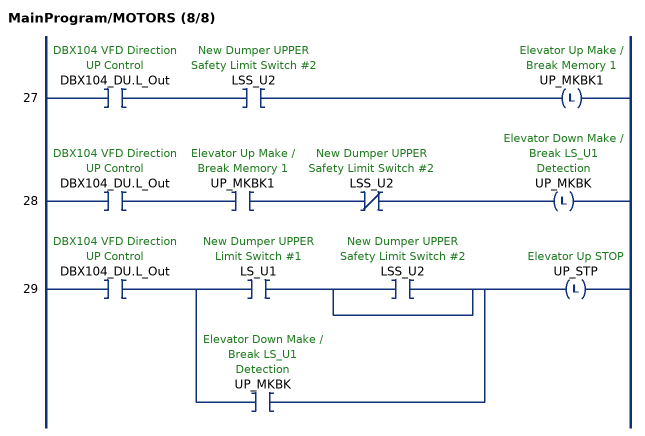
   27: XIC(DBX104_DU.L_Out)XIC(LSS_U2)OTL(UP_MKBK1);
   28: XIC(DBX104_DU.L_Out)XIC(UP_MKBK1)XIO(LSS_U2)OTL(UP_MKBK);
   29: XIC(DBX104_DU.L_Out)[XIC(LS_U1) [XIC(LSS_U2) ,] ,XIC(UP_MKBK) ]OTL(UP_STP);
END_ROUTINE
